(* IEC 61131-3 sources: PortalRobot/Portal_robot/Device/application (part 3) *)

(* ---- PLC_PRG.ReadHmiCommands.st ---- *)
METHOD PRIVATE ReadHmiCommands

// --- BEGIN IMPLEMENTATION ---

// Request counters belong to gateway; pulses and acknowledgements belong to PLC.
udiHmiCommandNowMs := TIME_TO_UDINT(TIME());
GVL_HMI.udiHmiCommandClockMs := udiHmiCommandNowMs;
FOR uiHmiCommandIndex := UINT#1 TO UINT#121 DO
	axHmiCommandConsumed[uiHmiCommandIndex] := FALSE;
	axHmiCommandPulse[uiHmiCommandIndex] := FALSE;
	// Mandatory low scan rearms every existing R_TRIG, including scenario events.
	IF NOT axHmiCommandWasHigh[uiHmiCommandIndex] THEN
		IF axHmiInternalPulse[uiHmiCommandIndex] THEN
			axHmiCommandPulse[uiHmiCommandIndex] := TRUE;
			axHmiInternalPulse[uiHmiCommandIndex] := FALSE;
		ELSE
			audiHmiCommandSnapshot[uiHmiCommandIndex] := GVL_HMI.audiHmiCommandSeq[uiHmiCommandIndex];
			IF (audiHmiCommandSnapshot[uiHmiCommandIndex] <> UDINT#0)
			AND (audiHmiCommandSnapshot[uiHmiCommandIndex] <> GVL_HMI.audiHmiCommandAckSeq[uiHmiCommandIndex]) THEN
				axHmiCommandConsumed[uiHmiCommandIndex] := TRUE;
				IF IsHmiCommandFresh(udiIssuedAtMs := GVL_HMI.audiHmiCommandIssuedAtMs[uiHmiCommandIndex]) THEN
					axHmiCommandPulse[uiHmiCommandIndex] := TRUE;
					GVL_HMI.auiHmiCommandResult[uiHmiCommandIndex] := UINT#1;
				ELSE
					GVL_HMI.auiHmiCommandResult[uiHmiCommandIndex] := UINT#2;
				END_IF;
			END_IF;
		END_IF;
	END_IF;
	axHmiCommandWasHigh[uiHmiCommandIndex] := axHmiCommandPulse[uiHmiCommandIndex];
END_FOR;

// Stable wire IDs; command-contract.mjs and static tests enforce this mapping.
GVL_HMI.xCellEnable := axHmiCommandPulse[1];
GVL_HMI.xCellDisable := axHmiCommandPulse[2];
GVL_HMI.xCellStart := axHmiCommandPulse[3];
GVL_HMI.xCellStop := axHmiCommandPulse[4];
GVL_HMI.xCellReset := axHmiCommandPulse[5];
GVL_HMI.xSafetyRelayReset := axHmiCommandPulse[6];
GVL_HMI.xCellOperatorCancel := axHmiCommandPulse[7];
GVL_HMI.xAlarmResetWarnings := axHmiCommandPulse[8];
GVL_HMI.xModbusSettingsApply := axHmiCommandPulse[9];
GVL_HMI.stMultiType.Command.xAutoDistribute := axHmiCommandPulse[10];
GVL_HMI.xSimAxisGroupError := axHmiCommandPulse[11];
GVL_HMI.xSimRobotWrongAction := axHmiCommandPulse[12];
GVL_HMI.xSimCellBothGrippers := axHmiCommandPulse[13];
GVL_HMI.xSimPointXOutOfLimit := axHmiCommandPulse[14];
GVL_HMI.xSimPointYOutOfLimit := axHmiCommandPulse[15];
GVL_HMI.xSimPointZOutOfLimit := axHmiCommandPulse[16];
GVL_HMI.xSimPointInvalidVelocity := axHmiCommandPulse[17];
GVL_HMI.xSimMagazineWrongOperation := axHmiCommandPulse[18];
GVL_HMI.xSimMagazineNoBlank := axHmiCommandPulse[19];
GVL_HMI.xSimMagazineNoFreeSlot := axHmiCommandPulse[20];
GVL_HMI.xSimMagazineInvalidSlot := axHmiCommandPulse[21];
GVL_HMI.xSimMagazineSlotContent := axHmiCommandPulse[22];
GVL_HMI.xSimMagazineGeometry := axHmiCommandPulse[23];
GVL_HMI.xRobotDrivesEnable := axHmiCommandPulse[24];
GVL_HMI.xRobotDrivesDisable := axHmiCommandPulse[25];
GVL_HMI.xRobotStop := axHmiCommandPulse[26];
GVL_HMI.xRobotReset := axHmiCommandPulse[27];
GVL_HMI.xTestEnvironmentApply := axHmiCommandPulse[28];
GVL_HMI.xTestSpeedProfileApply := axHmiCommandPulse[29];
GVL_HMI.xTestScenarioApply := axHmiCommandPulse[30];
GVL_HMI.xPointCheckStop := axHmiCommandPulse[31];
GVL_HMI.xRobotManualExecute := axHmiCommandPulse[32];
GVL_HMI.stMultiType.Command.xSetTypeCount := axHmiCommandPulse[33];
GVL_HMI.xCellOperatorChoice := axHmiCommandPulse[34];
GVL_HMI.stMultiType.Command.xSetMachineType := axHmiCommandPulse[35];
GVL_HMI.xRobotControlModeApply := axHmiCommandPulse[36];
GVL_HMI.stMultiType.Command.xSetSlotType := axHmiCommandPulse[37];
GVL_HMI.astAxisHmiCommand[1].xHome := axHmiCommandPulse[38];
GVL_HMI.astAxisHmiCommand[1].xMoveAbsolute := axHmiCommandPulse[39];
GVL_HMI.astAxisHmiCommand[1].xMoveRelative := axHmiCommandPulse[40];
GVL_HMI.axSimAxisJogConflict[1] := axHmiCommandPulse[41];
GVL_HMI.axMachineSimReset[1] := axHmiCommandPulse[42];
GVL_HMI.axMachineEnable[1] := axHmiCommandPulse[43];
GVL_HMI.axMachineDisable[1] := axHmiCommandPulse[44];
GVL_HMI.axMachineReset[1] := axHmiCommandPulse[45];
GVL_HMI.axMachineSetBlank[1] := axHmiCommandPulse[46];
GVL_HMI.axMachineSetDetail[1] := axHmiCommandPulse[47];
GVL_HMI.axMachineAcceptDoor[1] := axHmiCommandPulse[48];
GVL_HMI.axMachineRejectDoor[1] := axHmiCommandPulse[49];
GVL_HMI.axMachineAcceptRun[1] := axHmiCommandPulse[50];
GVL_HMI.axMachineRejectRun[1] := axHmiCommandPulse[51];
GVL_HMI.axMachineManualSafetyDoorOpen[1] := axHmiCommandPulse[52];
GVL_HMI.axMachineManualSafetyDoorClose[1] := axHmiCommandPulse[53];
GVL_HMI.axMachineManualHatchOpen[1] := axHmiCommandPulse[54];
GVL_HMI.axMachineManualHatchClose[1] := axHmiCommandPulse[55];
GVL_HMI.axMachineManualHatchUnlock[1] := axHmiCommandPulse[56];
GVL_HMI.axMachineManualHatchLock[1] := axHmiCommandPulse[57];
GVL_HMI.axMachineManualChuckOpen[1] := axHmiCommandPulse[58];
GVL_HMI.axMachineManualChuckClose[1] := axHmiCommandPulse[59];
GVL_HMI.astAxisHmiCommand[2].xHome := axHmiCommandPulse[60];
GVL_HMI.astAxisHmiCommand[2].xMoveAbsolute := axHmiCommandPulse[61];
GVL_HMI.astAxisHmiCommand[2].xMoveRelative := axHmiCommandPulse[62];
GVL_HMI.axSimAxisJogConflict[2] := axHmiCommandPulse[63];
GVL_HMI.axMachineSimReset[2] := axHmiCommandPulse[64];
GVL_HMI.axMachineEnable[2] := axHmiCommandPulse[65];
GVL_HMI.axMachineDisable[2] := axHmiCommandPulse[66];
GVL_HMI.axMachineReset[2] := axHmiCommandPulse[67];
GVL_HMI.axMachineSetBlank[2] := axHmiCommandPulse[68];
GVL_HMI.axMachineSetDetail[2] := axHmiCommandPulse[69];
GVL_HMI.axMachineAcceptDoor[2] := axHmiCommandPulse[70];
GVL_HMI.axMachineRejectDoor[2] := axHmiCommandPulse[71];
GVL_HMI.axMachineAcceptRun[2] := axHmiCommandPulse[72];
GVL_HMI.axMachineRejectRun[2] := axHmiCommandPulse[73];
GVL_HMI.axMachineManualSafetyDoorOpen[2] := axHmiCommandPulse[74];
GVL_HMI.axMachineManualSafetyDoorClose[2] := axHmiCommandPulse[75];
GVL_HMI.axMachineManualHatchOpen[2] := axHmiCommandPulse[76];
GVL_HMI.axMachineManualHatchClose[2] := axHmiCommandPulse[77];
GVL_HMI.axMachineManualHatchUnlock[2] := axHmiCommandPulse[78];
GVL_HMI.axMachineManualHatchLock[2] := axHmiCommandPulse[79];
GVL_HMI.axMachineManualChuckOpen[2] := axHmiCommandPulse[80];
GVL_HMI.axMachineManualChuckClose[2] := axHmiCommandPulse[81];
GVL_HMI.astAxisHmiCommand[3].xHome := axHmiCommandPulse[82];
GVL_HMI.astAxisHmiCommand[3].xMoveAbsolute := axHmiCommandPulse[83];
GVL_HMI.astAxisHmiCommand[3].xMoveRelative := axHmiCommandPulse[84];
GVL_HMI.axSimAxisJogConflict[3] := axHmiCommandPulse[85];
GVL_HMI.axMachineSimReset[3] := axHmiCommandPulse[86];
GVL_HMI.axMachineEnable[3] := axHmiCommandPulse[87];
GVL_HMI.axMachineDisable[3] := axHmiCommandPulse[88];
GVL_HMI.axMachineReset[3] := axHmiCommandPulse[89];
GVL_HMI.axMachineSetBlank[3] := axHmiCommandPulse[90];
GVL_HMI.axMachineSetDetail[3] := axHmiCommandPulse[91];
GVL_HMI.axMachineAcceptDoor[3] := axHmiCommandPulse[92];
GVL_HMI.axMachineRejectDoor[3] := axHmiCommandPulse[93];
GVL_HMI.axMachineAcceptRun[3] := axHmiCommandPulse[94];
GVL_HMI.axMachineRejectRun[3] := axHmiCommandPulse[95];
GVL_HMI.axMachineManualSafetyDoorOpen[3] := axHmiCommandPulse[96];
GVL_HMI.axMachineManualSafetyDoorClose[3] := axHmiCommandPulse[97];
GVL_HMI.axMachineManualHatchOpen[3] := axHmiCommandPulse[98];
GVL_HMI.axMachineManualHatchClose[3] := axHmiCommandPulse[99];
GVL_HMI.axMachineManualHatchUnlock[3] := axHmiCommandPulse[100];
GVL_HMI.axMachineManualHatchLock[3] := axHmiCommandPulse[101];
GVL_HMI.axMachineManualChuckOpen[3] := axHmiCommandPulse[102];
GVL_HMI.axMachineManualChuckClose[3] := axHmiCommandPulse[103];
GVL_HMI.astMagazineCommand[1].xEnable := axHmiCommandPulse[104];
GVL_HMI.astMagazineCommand[1].xDisable := axHmiCommandPulse[105];
GVL_HMI.astMagazineCommand[1].xStop := axHmiCommandPulse[106];
GVL_HMI.astMagazineCommand[1].xReset := axHmiCommandPulse[107];
GVL_HMI.astMagazineCommand[1].xFill := axHmiCommandPulse[108];
GVL_HMI.astMagazineCommand[1].xClear := axHmiCommandPulse[109];
GVL_HMI.astMagazineCommand[1].xApplySlot := axHmiCommandPulse[110];
GVL_HMI.astMagazineCommand[1].xApplyPitchX := axHmiCommandPulse[111];
GVL_HMI.astMagazineCommand[1].xApplyPitchY := axHmiCommandPulse[112];
GVL_HMI.astMagazineCommand[2].xEnable := axHmiCommandPulse[113];
GVL_HMI.astMagazineCommand[2].xDisable := axHmiCommandPulse[114];
GVL_HMI.astMagazineCommand[2].xStop := axHmiCommandPulse[115];
GVL_HMI.astMagazineCommand[2].xReset := axHmiCommandPulse[116];
GVL_HMI.astMagazineCommand[2].xFill := axHmiCommandPulse[117];
GVL_HMI.astMagazineCommand[2].xClear := axHmiCommandPulse[118];
GVL_HMI.astMagazineCommand[2].xApplySlot := axHmiCommandPulse[119];
GVL_HMI.astMagazineCommand[2].xApplyPitchX := axHmiCommandPulse[120];
GVL_HMI.astMagazineCommand[2].xApplyPitchY := axHmiCommandPulse[121];

(* ---- PLC_PRG.ReadHmiInputs.st ---- *)
METHOD PRIVATE ReadHmiInputs

// --- BEGIN IMPLEMENTATION ---

// HMI обязана поддерживать heartbeat. При потере связи PLC снимает только
// расширенные ручные команды; технологические проверки ниже остаются в PLC.
tonHmiWatchdog(
	IN := GVL_HMI.udiHmiHeartbeat = udiLastHmiHeartbeat,
	PT := T#2S
);
IF GVL_HMI.udiHmiHeartbeat <> udiLastHmiHeartbeat THEN
	udiLastHmiHeartbeat := GVL_HMI.udiHmiHeartbeat;
END_IF;
xHmiConnectionAlive := NOT tonHmiWatchdog.Q;

// Мобильная аренда отделена от общего HMI heartbeat. Gateway может быть жив,
// но движение обязано остановиться, если телефон перестал подтверждать аренду.
rtMobileMotionStart(CLK := GVL_HMI.xMobileMotionActive);
tonMobileMotionWatchdog(
	IN := GVL_HMI.xMobileMotionActive
		AND (GVL_HMI.udiMobileMotionHeartbeat = udiLastMobileMotionHeartbeat),
	PT := T#2S
);
IF GVL_HMI.udiMobileMotionHeartbeat <> udiLastMobileMotionHeartbeat THEN
	udiLastMobileMotionHeartbeat := GVL_HMI.udiMobileMotionHeartbeat;
END_IF;
IF rtMobileMotionStart.Q THEN
	xMobileMotionLeaseActive := TRUE;
	rMobileMotionSpeedLimitPercent := LIMIT(
		REAL#0.1,
		GVL_CELL_SETTINGS.rPointCheckSpeedPercent,
		REAL#100.0
	);
END_IF;
IF xMobileMotionLeaseActive THEN
	// Во время аренды лимит разрешено только уменьшать. Повышение настройки
	// применяется уже к следующему мобильному движению.
	rMobileMotionSpeedLimitPercent := MIN(
		rMobileMotionSpeedLimitPercent,
		LIMIT(REAL#0.1, GVL_CELL_SETTINGS.rPointCheckSpeedPercent, REAL#100.0)
	);
END_IF;
xMobileMotionConnectionAlive := GVL_HMI.xMobileMotionActive
	AND NOT tonMobileMotionWatchdog.Q;
xMobileMotionStopRequest := xMobileMotionLeaseActive
	AND (NOT GVL_HMI.xMobileMotionActive
		OR NOT xMobileMotionConnectionAlive
		OR NOT xHmiConnectionAlive);
IF xMobileMotionStopRequest THEN
	// Сбрасываем вход аренды в PLC: восстановление сети не может само возобновить ход.
	GVL_HMI.xMobileMotionActive := FALSE;
	FOR uiMachine := 1 TO 3 DO
		GVL_HMI.astAxisHmiCommand[uiMachine].xJogPositive := FALSE;
		GVL_HMI.astAxisHmiCommand[uiMachine].xJogNegative := FALSE;
	END_FOR;
END_IF;
GVL_HMI.xMobileMotionLeaseAlive := xMobileMotionLeaseActive
	AND xMobileMotionConnectionAlive
	AND NOT xMobileMotionStopRequest;
GVL_HMI.rMobileMotionAppliedSpeedPercent := rMobileMotionSpeedLimitPercent;

xPointCheckRequest := FALSE;
tonPointCheckWatchdog(IN := GVL_HMI.udiPointCheckHeartbeat = udiLastPointCheckHeartbeat, PT := T#2S);
IF GVL_HMI.udiPointCheckHeartbeat <> udiLastPointCheckHeartbeat THEN
	udiLastPointCheckHeartbeat := GVL_HMI.udiPointCheckHeartbeat;
END_IF;
xPointCheckConnectionAlive := (udiLastPointCheckHeartbeat <> UDINT#0) AND NOT tonPointCheckWatchdog.Q;
xPointCheckStopRequest := xPointCheckActive AND (GVL_HMI.xPointCheckStop
	OR NOT xPointCheckConnectionAlive OR NOT xHmiConnectionAlive);
// Stop is a PLC-owned one-scan event; its request counter is never cleared here.

IF GVL_HMI.rRobotManualSpeedPercent < REAL#0.1 THEN
	GVL_HMI.rRobotManualSpeedPercent := REAL#0.1;
ELSIF GVL_HMI.rRobotManualSpeedPercent > REAL#100.0 THEN
	GVL_HMI.rRobotManualSpeedPercent := REAL#100.0;
END_IF;
IF (GVL_HMI.lrRobotManualStep <> 0.1)
AND (GVL_HMI.lrRobotManualStep <> 1.0)
AND (GVL_HMI.lrRobotManualStep <> 10.0)
AND (GVL_HMI.lrRobotManualStep <> 100.0) THEN
	GVL_HMI.lrRobotManualStep := 1.0;
END_IF;

IF NOT xHmiConnectionAlive THEN
	FOR uiMachine := 1 TO 3 DO
		GVL_HMI.astAxisHmiCommand[uiMachine].xJogPositive := FALSE;
		GVL_HMI.astAxisHmiCommand[uiMachine].xJogNegative := FALSE;
		GVL_HMI.astAxisHmiCommand[uiMachine].xHome := FALSE;
		GVL_HMI.astAxisHmiCommand[uiMachine].xMoveAbsolute := FALSE;
		GVL_HMI.astAxisHmiCommand[uiMachine].xMoveRelative := FALSE;
	END_FOR;
	FOR uiMagazine := UINT#1 TO UINT#2 DO
		GVL_HMI.astMagazineCommand[uiMagazine].xStop := FALSE;
	END_FOR;
	GVL_HMI.xRobotManualExecute := FALSE;
END_IF;

// Глобальные команды ячейки поступают через единый интерфейс HMI.
GVL_CELL_CONTROL.xEnable := GVL_HMI.xCellEnable;
GVL_CELL_CONTROL.xDisable := GVL_HMI.xCellDisable;
GVL_CELL_CONTROL.xStart := GVL_HMI.xCellStart;
GVL_CELL_CONTROL.xStop := GVL_HMI.xCellStop;
// Необработанный общий импульс передаётся всем владельцам аварий.
// Каждый функциональный блок самостоятельно проверяет возможность сброса.
GVL_CELL_CONTROL.xReset := GVL_HMI.xCellReset;
// Режим хранит PLC. Новая транзакция применяется в RunSafety после чтения
// актуальных входов безопасности; PublishHmi не пишет в буфер запроса.
GVL_ALARM.Command.xResetWarnings := GVL_HMI.xAlarmResetWarnings;

// Режим инъекции ошибок включается отдельным переключателем страницы CELL_SETTINGS.
GVL_CELL_SETTINGS.xErrorSimulationEnabled := GVL_HMI.xErrorSimulationEnable;

// Ползунок меняет только запрошенное значение. Отдельный FB применяет его к
// таймерам и Dynamic Limits безопасной транзакцией перед следующим тестом.
GVL_CELL_SETTINGS.xSimulationAccelerationChangeAllowed :=
	xHmiConnectionAlive
	AND NOT GVL_CELL_CONTROL.xGlobalError;

IF GVL_CELL_SETTINGS.xSimulationAccelerationChangeAllowed THEN
	GVL_CELL_SETTINGS.xSimulationAccelerationEnable := GVL_HMI.xSimulationAccelerationEnable;
	GVL_CELL_SETTINGS.uiSimulationTimeFactor := GVL_HMI.uiSimulationTimeFactor;
	IF GVL_CELL_SETTINGS.uiSimulationTimeFactor < UINT#1 THEN
		GVL_CELL_SETTINGS.uiSimulationTimeFactor := UINT#1;
	ELSIF GVL_CELL_SETTINGS.uiSimulationTimeFactor > UINT#100 THEN
		GVL_CELL_SETTINGS.uiSimulationTimeFactor := UINT#100;
	END_IF;
ELSE
	// При потере разрешения сохраняем последнее принятое требование.
	GVL_HMI.xSimulationAccelerationEnable := GVL_CELL_SETTINGS.xSimulationAccelerationActive;
	GVL_HMI.uiSimulationTimeFactor := GVL_CELL_SETTINGS.uiSimulationTimeFactor;
END_IF;

// Общие технологические TIMEOUT и допуски HOME принимаются только при полностью
// остановленной ячейке. Координатами HOME_SAFETY владеет редактор точек ниже.
GVL_CELL_SETTINGS.xCellSettingsChangeAllowed :=
	xHmiConnectionAlive
	AND NOT GVL_CELL_MANAGER.Status.xRunning
	AND NOT GVL_HMI.xModbusMode
	AND NOT GVL_CELL_CONTROL.xGlobalError
	AND NOT GVL_AXIS.arrAxis[1].Status.xMotionBusy
	AND NOT GVL_AXIS.arrAxis[2].Status.xMotionBusy
	AND NOT GVL_AXIS.arrAxis[3].Status.xMotionBusy
	AND NOT GVL_AXIS_GROUP.AxisGroup.Command.xMoveDirect
	AND NOT GVL_AXIS_GROUP.AxisGroup.Command.xMoveLinear
	AND NOT GVL_ROBOT.Status.xBusy;

// Independent requested value; publication cannot overwrite an incoming write.
xCellSettingRejected := FALSE;
udiCellSettingSnapshot := GVL_HMI.udiCellSettingCommandSeq;
IF (udiCellSettingSnapshot <> UDINT#0)
AND (udiCellSettingSnapshot <> GVL_HMI.udiCellSettingAckSeq) THEN
	GVL_HMI.uiCellSettingResult := UINT#3;
	IF NOT IsHmiCommandFresh(udiIssuedAtMs := GVL_HMI.udiCellSettingIssuedAtMs) THEN
		GVL_HMI.uiCellSettingResult := UINT#4; // Expired: never apply later
	ELSIF NOT GVL_CELL_SETTINGS.xCellSettingsChangeAllowed
	OR ((GVL_HMI.uiCellSettingIndex = UINT#4) AND xPointCheckActive) THEN
		GVL_HMI.uiCellSettingResult := UINT#2;
	ELSE
		CASE GVL_HMI.uiCellSettingIndex OF
			UINT#1:
				IF (GVL_HMI.lrCellSettingRequest >= 0.1) AND (GVL_HMI.lrCellSettingRequest <= 1000.0) THEN
					GVL_CELL_SETTINGS.lrSafetyHomeToleranceX := GVL_HMI.lrCellSettingRequest;
					GVL_HMI.uiCellSettingResult := UINT#1;
				END_IF;
			UINT#2:
				IF (GVL_HMI.lrCellSettingRequest >= 0.1) AND (GVL_HMI.lrCellSettingRequest <= 1000.0) THEN
					GVL_CELL_SETTINGS.lrSafetyHomeToleranceY := GVL_HMI.lrCellSettingRequest;
					GVL_HMI.uiCellSettingResult := UINT#1;
				END_IF;
			UINT#3:
				IF (GVL_HMI.lrCellSettingRequest >= 0.1) AND (GVL_HMI.lrCellSettingRequest <= 1000.0) THEN
					GVL_CELL_SETTINGS.lrSafetyHomeToleranceZ := GVL_HMI.lrCellSettingRequest;
					GVL_HMI.uiCellSettingResult := UINT#1;
				END_IF;
			UINT#4:
				IF (GVL_HMI.lrCellSettingRequest >= 0.1) AND (GVL_HMI.lrCellSettingRequest <= 100.0) THEN
					GVL_CELL_SETTINGS.rPointCheckSpeedPercent := LREAL_TO_REAL(GVL_HMI.lrCellSettingRequest);
					GVL_HMI.uiCellSettingResult := UINT#1;
				END_IF;
			UINT#5:
				IF (GVL_HMI.lrCellSettingRequest >= 1000.0) AND (GVL_HMI.lrCellSettingRequest <= 600000.0) THEN
					GVL_CELL_SETTINGS.stMachineTimeouts.tRobotMove := UDINT_TO_TIME(LREAL_TO_UDINT(GVL_HMI.lrCellSettingRequest));
					GVL_HMI.uiCellSettingResult := UINT#1;
				END_IF;
			UINT#6:
				IF (GVL_HMI.lrCellSettingRequest >= 1000.0) AND (GVL_HMI.lrCellSettingRequest <= 600000.0) THEN
					GVL_CELL_SETTINGS.stMachineTimeouts.tRobotAction := UDINT_TO_TIME(LREAL_TO_UDINT(GVL_HMI.lrCellSettingRequest));
					GVL_HMI.uiCellSettingResult := UINT#1;
				END_IF;
			UINT#7:
				IF (GVL_HMI.lrCellSettingRequest >= 1000.0) AND (GVL_HMI.lrCellSettingRequest <= 600000.0) THEN
					GVL_CELL_SETTINGS.stMachineTimeouts.tRobotRelease := UDINT_TO_TIME(LREAL_TO_UDINT(GVL_HMI.lrCellSettingRequest));
					GVL_HMI.uiCellSettingResult := UINT#1;
				END_IF;
			UINT#8:
				IF (GVL_HMI.lrCellSettingRequest >= 1000.0) AND (GVL_HMI.lrCellSettingRequest <= 600000.0) THEN
					GVL_CELL_SETTINGS.stMachineTimeouts.tDoorOpen := UDINT_TO_TIME(LREAL_TO_UDINT(GVL_HMI.lrCellSettingRequest));
					GVL_HMI.uiCellSettingResult := UINT#1;
				END_IF;
			UINT#9:
				IF (GVL_HMI.lrCellSettingRequest >= 1000.0) AND (GVL_HMI.lrCellSettingRequest <= 600000.0) THEN
					GVL_CELL_SETTINGS.stMachineTimeouts.tDoorClose := UDINT_TO_TIME(LREAL_TO_UDINT(GVL_HMI.lrCellSettingRequest));
					GVL_HMI.uiCellSettingResult := UINT#1;
				END_IF;
			UINT#10:
				IF (GVL_HMI.lrCellSettingRequest >= 1000.0) AND (GVL_HMI.lrCellSettingRequest <= 600000.0) THEN
					GVL_CELL_SETTINGS.stMachineTimeouts.tHatchUnlock := UDINT_TO_TIME(LREAL_TO_UDINT(GVL_HMI.lrCellSettingRequest));
					GVL_HMI.uiCellSettingResult := UINT#1;
				END_IF;
			UINT#11:
				IF (GVL_HMI.lrCellSettingRequest >= 1000.0) AND (GVL_HMI.lrCellSettingRequest <= 600000.0) THEN
					GVL_CELL_SETTINGS.stMachineTimeouts.tChuckOpen := UDINT_TO_TIME(LREAL_TO_UDINT(GVL_HMI.lrCellSettingRequest));
					GVL_HMI.uiCellSettingResult := UINT#1;
				END_IF;
			UINT#12:
				IF (GVL_HMI.lrCellSettingRequest >= 1000.0) AND (GVL_HMI.lrCellSettingRequest <= 600000.0) THEN
					GVL_CELL_SETTINGS.stMachineTimeouts.tChuckClose := UDINT_TO_TIME(LREAL_TO_UDINT(GVL_HMI.lrCellSettingRequest));
					GVL_HMI.uiCellSettingResult := UINT#1;
				END_IF;
			UINT#13:
				IF (GVL_HMI.lrCellSettingRequest >= 1000.0) AND (GVL_HMI.lrCellSettingRequest <= 600000.0) THEN
					GVL_CELL_SETTINGS.stMachineTimeouts.tCycleStart := UDINT_TO_TIME(LREAL_TO_UDINT(GVL_HMI.lrCellSettingRequest));
					GVL_HMI.uiCellSettingResult := UINT#1;
				END_IF;
		END_CASE;
	END_IF;
	xCellSettingRejected := GVL_HMI.uiCellSettingResult <> UINT#1;
END_IF;

// =============================================================================
// Транзакционный редактор 12 фиксированных инженерных точек
// =============================================================================
xPointEditorAllHomed := GVL_AXIS.arrAxis[1].Status.xHomed
	AND GVL_AXIS.arrAxis[2].Status.xHomed
	AND GVL_AXIS.arrAxis[3].Status.xHomed;
xPointEditorBaseAllowed := xHmiConnectionAlive
	AND NOT xPointCheckActive
	AND GVL_CELL_CONTROL.xManual
	AND NOT GVL_HMI.xModbusMode
	AND NOT GVL_CELL_MANAGER.Status.xRunning
	AND NOT GVL_CELL_CONTROL.xGlobalError
	AND NOT GVL_ROBOT.Status.xBusy
	AND NOT xMotionBusy
	AND NOT xDriveError
	AND NOT GVL_MOTION_MANAGER.stMotionManager.Status.xError
	AND xPointEditorAllHomed
	AND GVL_AXIS_GROUP.AxisGroup.Status.xPositionValid;
GVL_HMI.xPointEditorCaptureAllowed := xPointEditorBaseAllowed;
GVL_HMI.xPointEditorSaveAllowed := xPointEditorBaseAllowed
	AND GVL_POINT_MANAGER.PointManager.Diag.xXLimitValid
	AND GVL_POINT_MANAGER.PointManager.Diag.xYLimitValid
	AND GVL_POINT_MANAGER.PointManager.Diag.xZLimitValid;

IF (GVL_HMI.udiPointEditorCommandSeq <> UDINT#0)
AND (GVL_HMI.udiPointEditorCommandSeq <> udiLastPointEditorCommandSeq) THEN
	udiLastPointEditorCommandSeq := GVL_HMI.udiPointEditorCommandSeq;
	GVL_HMI.uiPointEditorResult := UINT#2;
	GVL_HMI.uiPointEditorRejectReason := UINT#0;
	xPointEditorRequestValid := FALSE;
	xPointEditorMagazinePoint := FALSE;
	ePointEditorName := E_POINT_NAME.NONE;
	uiPointStorageIndex := UINT#0;

	CASE GVL_HMI.uiPointEditorIndex OF
		UINT#1: ePointEditorName := E_POINT_NAME.MACHINE_1_ABOVE; uiPointStorageIndex := UINT#1;
		UINT#2: ePointEditorName := E_POINT_NAME.MACHINE_1_CHUCK_APROACH; uiPointStorageIndex := UINT#3;
		UINT#3: ePointEditorName := E_POINT_NAME.MACHINE_1_CHUCK_POSITION; uiPointStorageIndex := UINT#4;
		UINT#4: ePointEditorName := E_POINT_NAME.MACHINE_2_ABOVE; uiPointStorageIndex := UINT#5;
		UINT#5: ePointEditorName := E_POINT_NAME.MACHINE_2_CHUCK_APROACH; uiPointStorageIndex := UINT#7;
		UINT#6: ePointEditorName := E_POINT_NAME.MACHINE_2_CHUCK_POSITION; uiPointStorageIndex := UINT#8;
		UINT#7: ePointEditorName := E_POINT_NAME.MACHINE_3_ABOVE; uiPointStorageIndex := UINT#9;
		UINT#8: ePointEditorName := E_POINT_NAME.MACHINE_3_CHUCK_APROACH; uiPointStorageIndex := UINT#11;
		UINT#9: ePointEditorName := E_POINT_NAME.MACHINE_3_CHUCK_POSITION; uiPointStorageIndex := UINT#12;
		UINT#10: ePointEditorName := E_POINT_NAME.HOME_SAFETY; uiPointStorageIndex := UINT#13;
		UINT#11: ePointEditorName := E_POINT_NAME.MAGAZINE_1_DETAIL; uiPointStorageIndex := UINT#14;
		UINT#12: ePointEditorName := E_POINT_NAME.MAGAZINE_2_DETAIL; uiPointStorageIndex := UINT#15;
	END_CASE;
	xPointEditorRequestValid := (ePointEditorName <> E_POINT_NAME.NONE)
		AND (uiPointStorageIndex <> UINT#0);
	xPointEditorMagazinePoint := (ePointEditorName = E_POINT_NAME.MAGAZINE_1_DETAIL)
		OR (ePointEditorName = E_POINT_NAME.MAGAZINE_2_DETAIL);

	IF (GVL_HMI.uiPointEditorCommand <> UINT#1)
	AND (GVL_HMI.uiPointEditorCommand <> UINT#2)
	AND (GVL_HMI.uiPointEditorCommand <> UINT#3) THEN
		GVL_HMI.uiPointEditorRejectReason := UINT#1; // Неизвестная команда
	ELSIF NOT xPointEditorRequestValid THEN
		GVL_HMI.uiPointEditorRejectReason := UINT#2; // Неверный индекс точки
	ELSIF NOT xHmiConnectionAlive THEN
		GVL_HMI.uiPointEditorRejectReason := UINT#3; // HMI offline
	ELSIF NOT GVL_CELL_CONTROL.xManual THEN
		GVL_HMI.uiPointEditorRejectReason := UINT#4; // Требуется ручной режим
	ELSIF GVL_HMI.xModbusMode THEN
		GVL_HMI.uiPointEditorRejectReason := UINT#5; // Требуется SoftMotion
	ELSIF GVL_CELL_MANAGER.Status.xRunning THEN
		GVL_HMI.uiPointEditorRejectReason := UINT#6; // Автоматический цикл выполняется
	ELSIF GVL_CELL_CONTROL.xGlobalError THEN
		GVL_HMI.uiPointEditorRejectReason := UINT#7; // Глобальная ошибка
	ELSIF GVL_ROBOT.Status.xBusy OR xPointCheckActive THEN
		GVL_HMI.uiPointEditorRejectReason := UINT#8; // Робот занят
	ELSIF xMotionBusy THEN
		GVL_HMI.uiPointEditorRejectReason := UINT#9; // Motion занят
	ELSIF xDriveError OR GVL_MOTION_MANAGER.stMotionManager.Status.xError THEN
		GVL_HMI.uiPointEditorRejectReason := UINT#10; // Ошибка оси или группы
	ELSIF NOT xPointEditorAllHomed THEN
		GVL_HMI.uiPointEditorRejectReason := UINT#11; // Не выполнен Home
	ELSIF NOT GVL_AXIS_GROUP.AxisGroup.Status.xPositionValid THEN
		GVL_HMI.uiPointEditorRejectReason := UINT#12; // Недостоверные координаты
	ELSIF (GVL_HMI.uiPointEditorCommand = UINT#2)
	AND (NOT GVL_POINT_MANAGER.PointManager.Diag.xXLimitValid
		OR NOT GVL_POINT_MANAGER.PointManager.Diag.xYLimitValid
		OR NOT GVL_POINT_MANAGER.PointManager.Diag.xZLimitValid) THEN
		GVL_HMI.uiPointEditorRejectReason := UINT#13; // Software limits недоступны
	ELSE
		IF GVL_HMI.uiPointEditorCommand = UINT#1 THEN
			// CAPTURE возвращает согласованный снимок одного PLC-цикла и не пишет Persistent.
			GVL_HMI.stPointEditorResultPoint.Name := '';
			GVL_HMI.stPointEditorResultPoint.X := GVL_AXIS_GROUP.AxisGroup.Status.ActualX;
			GVL_HMI.stPointEditorResultPoint.Y := GVL_AXIS_GROUP.AxisGroup.Status.ActualY;
			GVL_HMI.stPointEditorResultPoint.Z := GVL_AXIS_GROUP.AxisGroup.Status.ActualZ;
			GVL_HMI.stPointEditorResultPoint.MagazineSafeZ :=
				GVL_HMI.lrPointEditorDraftMagazineSafeZ;
			GVL_HMI.stPointEditorResultPoint.MagazineChangeZ :=
				GVL_HMI.lrPointEditorDraftMagazineChangeZ;
			GVL_HMI.stPointEditorResultPoint.SpeedFactor :=
				GVL_HMI.lrPointEditorDraftSpeedFactor;
			GVL_HMI.stPointEditorResultPoint.xConfigured := FALSE;
			GVL_HMI.uiPointEditorResult := UINT#1;
		ELSIF GVL_HMI.uiPointEditorCommand = UINT#3 THEN
			// CHECK никогда не сохраняет черновик. Сравнение защищает подтверждение
			// на телефоне от изменения точки другим редактором до запуска.
			IF NOT GVL_POINT.Points[ePointEditorName].xConfigured THEN
				GVL_HMI.uiPointEditorRejectReason := UINT#16;
			ELSIF (GVL_POINT.Points[ePointEditorName].X <> GVL_HMI.alrPointEditorDraftXYZ[1])
			OR (GVL_POINT.Points[ePointEditorName].Y <> GVL_HMI.alrPointEditorDraftXYZ[2])
			OR (GVL_POINT.Points[ePointEditorName].Z <> GVL_HMI.alrPointEditorDraftXYZ[3])
			OR (GVL_POINT.Points[ePointEditorName].SpeedFactor <> GVL_HMI.lrPointEditorDraftSpeedFactor)
			OR (xPointEditorMagazinePoint
				AND ((GVL_POINT.Points[ePointEditorName].MagazineSafeZ <>
					GVL_HMI.lrPointEditorDraftMagazineSafeZ)
				OR (GVL_POINT.Points[ePointEditorName].MagazineChangeZ <>
					GVL_HMI.lrPointEditorDraftMagazineChangeZ))) THEN
				GVL_HMI.uiPointEditorRejectReason := UINT#21;
			ELSE
				xPointCheckRequest := TRUE; // Финальное разрешение после RunMotion/RunCellControl
			END_IF;
		ELSE
			xPointEditorDraftValid :=
				(GVL_HMI.alrPointEditorDraftXYZ[1] >= alrRobotSoftwareMinPosition[1])
				AND (GVL_HMI.alrPointEditorDraftXYZ[1] <= alrRobotSoftwareMaxPosition[1])
				AND (GVL_HMI.alrPointEditorDraftXYZ[2] >= alrRobotSoftwareMinPosition[2])
				AND (GVL_HMI.alrPointEditorDraftXYZ[2] <= alrRobotSoftwareMaxPosition[2])
				AND (GVL_HMI.alrPointEditorDraftXYZ[3] >= alrRobotSoftwareMinPosition[3])
				AND (GVL_HMI.alrPointEditorDraftXYZ[3] <= alrRobotSoftwareMaxPosition[3]);
			IF NOT xPointEditorDraftValid THEN
				GVL_HMI.uiPointEditorRejectReason := UINT#14; // XYZ вне software limits
			ELSIF NOT ((GVL_HMI.lrPointEditorDraftSpeedFactor > 0.1)
			AND (GVL_HMI.lrPointEditorDraftSpeedFactor <= 1.0)) THEN
				GVL_HMI.uiPointEditorRejectReason := UINT#15; // Недопустимая скорость
			ELSIF xPointEditorMagazinePoint
			AND ((GVL_HMI.lrPointEditorDraftMagazineSafeZ < -LREAL#10000.0)
				OR (GVL_HMI.lrPointEditorDraftMagazineSafeZ > LREAL#10000.0)
				OR (GVL_HMI.lrPointEditorDraftMagazineChangeZ < -LREAL#10000.0)
				OR (GVL_HMI.lrPointEditorDraftMagazineChangeZ > LREAL#10000.0)) THEN
				GVL_HMI.uiPointEditorRejectReason := UINT#22; // Смещения магазина вне диапазона
			ELSE
				GVL_POINT.astRetainPoints[uiPointStorageIndex].Name := '';
				GVL_POINT.astRetainPoints[uiPointStorageIndex].X :=
					GVL_HMI.alrPointEditorDraftXYZ[1];
				GVL_POINT.astRetainPoints[uiPointStorageIndex].Y :=
					GVL_HMI.alrPointEditorDraftXYZ[2];
				GVL_POINT.astRetainPoints[uiPointStorageIndex].Z :=
					GVL_HMI.alrPointEditorDraftXYZ[3];
				IF xPointEditorMagazinePoint THEN
					GVL_POINT.astRetainPoints[uiPointStorageIndex].MagazineSafeZ :=
						GVL_HMI.lrPointEditorDraftMagazineSafeZ;
					GVL_POINT.astRetainPoints[uiPointStorageIndex].MagazineChangeZ :=
						GVL_HMI.lrPointEditorDraftMagazineChangeZ;
				ELSE
					GVL_POINT.astRetainPoints[uiPointStorageIndex].MagazineSafeZ := LREAL#0.0;
					GVL_POINT.astRetainPoints[uiPointStorageIndex].MagazineChangeZ := LREAL#0.0;
				END_IF;
				GVL_POINT.astRetainPoints[uiPointStorageIndex].SpeedFactor :=
					GVL_HMI.lrPointEditorDraftSpeedFactor;
				GVL_POINT.astRetainPoints[uiPointStorageIndex].xConfigured :=
					NOT xPointEditorMagazinePoint
					OR ((GVL_HMI.lrPointEditorDraftMagazineSafeZ <> LREAL#0.0)
						AND (GVL_HMI.lrPointEditorDraftMagazineChangeZ <> LREAL#0.0));
				GVL_POINT.Points[ePointEditorName] :=
					GVL_POINT.astRetainPoints[uiPointStorageIndex];
				GVL_HMI.stPointEditorResultPoint := GVL_POINT.Points[ePointEditorName];
				GVL_HMI.uiPointEditorResult := UINT#1;
			END_IF;
		END_IF;
	END_IF;

	IF (GVL_HMI.uiPointEditorResult <> UINT#1) AND NOT xPointCheckRequest THEN
		IF GVL_HMI.uiPointEditorCommand = UINT#3 THEN
			uiRobotInterfaceWarningCode := WRN_POINT_CHECK_REJECTED;
		ELSE
			uiRobotInterfaceWarningCode := WRN_POINT_EDIT_REJECTED;
		END_IF;
	END_IF;
	// Ack подтверждает обработку конкретной транзакции даже при отказе.
	IF NOT xPointCheckRequest THEN
		GVL_HMI.udiPointEditorAckSeq := GVL_HMI.udiPointEditorCommandSeq;
	END_IF;
END_IF;

// Плоский OPC UA-интерфейс HMI преобразуется в типизированные запросы FB.
FOR uiMachine := 1 TO 3 DO
	astMachineFaultRequest[uiMachine].xEnabled := GVL_CELL_SETTINGS.xErrorSimulationEnabled;
	astMachineFaultRequest[uiMachine].xReset := GVL_HMI.axMachineSimReset[uiMachine];
	astMachineFaultRequest[uiMachine].xMachineAlarm := GVL_HMI.axMachineSimAlarm[uiMachine];
	astMachineFaultRequest[uiMachine].xDoorFault := GVL_HMI.axMachineSimDoorFault[uiMachine];
	astMachineFaultRequest[uiMachine].xChuckFault := GVL_HMI.axMachineSimChuckFault[uiMachine];
	astMachineFaultRequest[uiMachine].xTimeoutRobotMove := GVL_HMI.axMachineTimeoutRobotMove[uiMachine];
	astMachineFaultRequest[uiMachine].xTimeoutRobotAction := GVL_HMI.axMachineTimeoutRobotAction[uiMachine];
	astMachineFaultRequest[uiMachine].xTimeoutRobotRelease := GVL_HMI.axMachineTimeoutRobotRelease[uiMachine];
	astMachineFaultRequest[uiMachine].xTimeoutDoorOpen := GVL_HMI.axMachineTimeoutDoorOpen[uiMachine];
	astMachineFaultRequest[uiMachine].xTimeoutDoorClose := GVL_HMI.axMachineTimeoutDoorClose[uiMachine];
	astMachineFaultRequest[uiMachine].xTimeoutHatchUnlock := GVL_HMI.axMachineTimeoutHatchUnlock[uiMachine];
	astMachineFaultRequest[uiMachine].xTimeoutChuckOpen := GVL_HMI.axMachineTimeoutChuckOpen[uiMachine];
	astMachineFaultRequest[uiMachine].xTimeoutChuckClose := GVL_HMI.axMachineTimeoutChuckClose[uiMachine];
	astMachineFaultRequest[uiMachine].xTimeoutCycleStart := GVL_HMI.axMachineTimeoutCycleStart[uiMachine];

	astAxisFaultRequest[uiMachine].xEnabled := GVL_CELL_SETTINGS.xErrorSimulationEnabled;
	astAxisFaultRequest[uiMachine].xJogConflict := GVL_HMI.axSimAxisJogConflict[uiMachine];
END_FOR;

stAxisGroupFaultRequest.xEnabled := GVL_CELL_SETTINGS.xErrorSimulationEnabled;
stAxisGroupFaultRequest.xExecute := GVL_HMI.xSimAxisGroupError;

stRobotFaultRequest.xEnabled := GVL_CELL_SETTINGS.xErrorSimulationEnabled;
stRobotFaultRequest.xWrongAction := GVL_HMI.xSimRobotWrongAction;
stRobotFaultRequest.stGripper.xEnabled := GVL_CELL_SETTINGS.xErrorSimulationEnabled;
stRobotFaultRequest.stGripper.xGripper1Fault := GVL_HMI.xSimGripper1Fault;
stRobotFaultRequest.stGripper.xGripper2Fault := GVL_HMI.xSimGripper2Fault;
stRobotFaultRequest.stGripper.xRotationFault := GVL_HMI.xSimGripperRotationFault;
stRobotFaultRequest.stGripper.xGlobalFault := GVL_HMI.xSimGripperGlobalFault;

stRobotFaultRequest.stPoint.xEnabled := GVL_CELL_SETTINGS.xErrorSimulationEnabled;
stRobotFaultRequest.stPoint.xXOutOfLimit := GVL_HMI.xSimPointXOutOfLimit;
stRobotFaultRequest.stPoint.xYOutOfLimit := GVL_HMI.xSimPointYOutOfLimit;
stRobotFaultRequest.stPoint.xZOutOfLimit := GVL_HMI.xSimPointZOutOfLimit;
stRobotFaultRequest.stPoint.xInvalidVelocity := GVL_HMI.xSimPointInvalidVelocity;

IF NOT GVL_CELL_SETTINGS.xErrorSimulationEnabled THEN
	adwTestMagazineFaultMask[1] := DWORD#0;
	adwTestMagazineFaultMask[2] := DWORD#0;
END_IF;
astMagazineFaultRequest[1].xEnabled := GVL_CELL_SETTINGS.xErrorSimulationEnabled;
astMagazineFaultRequest[1].xWrongOperation := GVL_HMI.xSimMagazineWrongOperation
	OR ((adwTestMagazineFaultMask[1] AND DWORD#16#0000_0001) <> DWORD#0);
astMagazineFaultRequest[1].xNoBlank := GVL_HMI.xSimMagazineNoBlank
	OR ((adwTestMagazineFaultMask[1] AND DWORD#16#0000_0002) <> DWORD#0);
astMagazineFaultRequest[1].xNoFreeSlot := GVL_HMI.xSimMagazineNoFreeSlot
	OR ((adwTestMagazineFaultMask[1] AND DWORD#16#0000_0004) <> DWORD#0);
astMagazineFaultRequest[1].xInvalidSlot := GVL_HMI.xSimMagazineInvalidSlot
	OR ((adwTestMagazineFaultMask[1] AND DWORD#16#0000_0008) <> DWORD#0);
astMagazineFaultRequest[1].xSlotContent := GVL_HMI.xSimMagazineSlotContent
	OR ((adwTestMagazineFaultMask[1] AND DWORD#16#0000_0010) <> DWORD#0);
astMagazineFaultRequest[1].xGeometry := GVL_HMI.xSimMagazineGeometry
	OR ((adwTestMagazineFaultMask[1] AND DWORD#16#0000_0020) <> DWORD#0);
astMagazineFaultRequest[2].xEnabled := GVL_CELL_SETTINGS.xErrorSimulationEnabled
	AND (adwTestMagazineFaultMask[2] <> DWORD#0);
astMagazineFaultRequest[2].xWrongOperation :=
	(adwTestMagazineFaultMask[2] AND DWORD#16#0000_0001) <> DWORD#0;
astMagazineFaultRequest[2].xNoBlank :=
	(adwTestMagazineFaultMask[2] AND DWORD#16#0000_0002) <> DWORD#0;
astMagazineFaultRequest[2].xNoFreeSlot :=
	(adwTestMagazineFaultMask[2] AND DWORD#16#0000_0004) <> DWORD#0;
astMagazineFaultRequest[2].xInvalidSlot :=
	(adwTestMagazineFaultMask[2] AND DWORD#16#0000_0008) <> DWORD#0;
astMagazineFaultRequest[2].xSlotContent :=
	(adwTestMagazineFaultMask[2] AND DWORD#16#0000_0010) <> DWORD#0;
astMagazineFaultRequest[2].xGeometry :=
	(adwTestMagazineFaultMask[2] AND DWORD#16#0000_0020) <> DWORD#0;

stCellFaultRequest.xEnabled := GVL_CELL_SETTINGS.xErrorSimulationEnabled;
stCellFaultRequest.xBothGrippers := GVL_HMI.xSimCellBothGrippers;

stSafetyFaultRequest.xEnabled := GVL_CELL_SETTINGS.xErrorSimulationEnabled;
FOR uiMachine := UINT#1 TO UINT#4 DO
	stSafetyFaultRequest.axEmergencyStopStation[uiMachine] :=
		GVL_HMI.axSimSafetyEmergencyStopStation[uiMachine];
	stSafetyFaultRequest.axDoorUnlocked[uiMachine] :=
		GVL_HMI.axSimSafetyDoorUnlocked[uiMachine];
END_FOR;
FOR uiMachine := UINT#1 TO UINT#2 DO
	stSafetyFaultRequest.axEmergencyStopCabinet[uiMachine] :=
		GVL_HMI.axSimSafetyEmergencyStopCabinet[uiMachine];
END_FOR;
stSafetyFaultRequest.xEmergencyStopMpg := GVL_HMI.xSimSafetyEmergencyStopMpg;
stSafetyFaultRequest.xPhaseRelayFault := GVL_HMI.xSimSafetyPhaseRelayFault;
stSafetyFaultRequest.xPressureRelayFault := GVL_HMI.xSimSafetyPressureRelayFault;
stSafetyFaultRequest.xSafetyRelayFault := GVL_HMI.xSimSafetyRelayFault;

(* ---- PLC_PRG.RunAlarms.st ---- *)
METHOD PRIVATE RunAlarms

// --- BEGIN IMPLEMENTATION ---

// Единая кнопка подсвечивается только тогда, когда существует хотя бы одна авария
// и каждый активный владелец общей команды готов принять тот же импульс сброса.
// Диагностические защёлки симуляторов станков сюда не входят: они обслуживаются
// отдельной командой «Сброс симулятора» на экране инъекций.
xAlarmResetRequired := GVL_CELL_MANAGER.Status.xError
	OR (CELL_SAFETY.Error.dwAlarmActive <> DWORD#0)
	OR GVL_ROBOT.Status.xError
	OR GVL_MACHINE.Status[1].xError
	OR GVL_MACHINE.Status[2].xError
	OR GVL_MACHINE.Status[3].xError
	OR GVL_MAGAZINE.astStatus[1].xError
	OR GVL_MAGAZINE.astStatus[2].xError
	OR (NOT GVL_HMI.xModbusMode AND GVL_AXIS.arrAxis[1].Status.xError)
	OR (NOT GVL_HMI.xModbusMode AND GVL_AXIS.arrAxis[2].Status.xError)
	OR (NOT GVL_HMI.xModbusMode AND GVL_AXIS.arrAxis[3].Status.xError)
	OR (NOT GVL_HMI.xModbusMode AND GVL_AXIS_GROUP.AxisGroup.Status.xLocalError)
	OR (NOT GVL_HMI.xModbusMode AND GVL_AXIS_GROUP.AxisGroup.Status.xLogicalError)
	OR (NOT GVL_HMI.xModbusMode AND GVL_AXIS_GROUP.AxisGroup.Status.xGroupError)
	OR (NOT GVL_HMI.xModbusMode AND (GVL_MOTION_MANAGER.stMotionManager.Error.dwAlarmActive <> DWORD#0))
	OR (NOT GVL_HMI.xModbusMode AND (GVL_POINT_MANAGER.PointManager.Error.dwAlarmActive <> DWORD#0))
	OR (NOT GVL_HMI.xModbusMode AND (GVL_ROBOT.GripperError.dwAlarmActive <> DWORD#0));

xAlarmResetAllowed := ((GVL_TWO_PALLET.uiMode = 0) OR ((NOT GVL_TWO_PALLET.astStatus[1].xError OR GVL_TWO_PALLET.astStatus[1].xResetAllowed) AND (NOT GVL_TWO_PALLET.astStatus[2].xError OR GVL_TWO_PALLET.astStatus[2].xResetAllowed))) AND xAlarmResetRequired
	AND (CELL_SAFETY.Error.dwAlarmActive = DWORD#0)
	AND (NOT GVL_CELL_MANAGER.Status.xError OR GVL_CELL_MANAGER.Status.xResetAllowed)
	AND (NOT GVL_ROBOT.Status.xError OR GVL_ROBOT.Status.xResetAllowed)
	AND (NOT GVL_MACHINE.Status[1].xError OR GVL_MACHINE.Status[1].xResetAllowed)
	AND (NOT GVL_MACHINE.Status[2].xError OR GVL_MACHINE.Status[2].xResetAllowed)
	AND (NOT GVL_MACHINE.Status[3].xError OR GVL_MACHINE.Status[3].xResetAllowed)
	AND (NOT GVL_MAGAZINE.astPartStatus[1].xError
		OR (GVL_MAGAZINE.astError[1].dwAlarmActive = DWORD#0)
		OR fbMagazine1.FaultStatus.xResetAllowed)
	AND (NOT GVL_MAGAZINE.astPartStatus[2].xError
		OR (GVL_MAGAZINE.astError[2].dwAlarmActive = DWORD#0)
		OR fbMagazine2.FaultStatus.xResetAllowed)
	AND (GVL_HMI.xModbusMode OR NOT GVL_AXIS.arrAxis[1].Status.xError OR AXIS_X.FaultStatus.xResetAllowed)
	AND (GVL_HMI.xModbusMode OR NOT GVL_AXIS.arrAxis[2].Status.xError OR AXIS_Y.FaultStatus.xResetAllowed)
	AND (GVL_HMI.xModbusMode OR NOT GVL_AXIS.arrAxis[3].Status.xError OR AXIS_Z.FaultStatus.xResetAllowed)
	AND (GVL_HMI.xModbusMode OR NOT (GVL_AXIS_GROUP.AxisGroup.Status.xLocalError
		OR GVL_AXIS_GROUP.AxisGroup.Status.xLogicalError
		OR GVL_AXIS_GROUP.AxisGroup.Status.xGroupError)
		OR GROUP_XYZ.FaultStatus.xResetAllowed)
	AND (GVL_HMI.xModbusMode OR (GVL_MOTION_MANAGER.stMotionManager.Error.dwAlarmActive = DWORD#0)
		OR GVL_ROBOT.Status.xResetAllowed)
	AND (GVL_HMI.xModbusMode OR (GVL_POINT_MANAGER.PointManager.Error.dwAlarmActive = DWORD#0)
		OR (GVL_ROBOT.Status.xResetAllowed AND ROBOT.FaultStatus.stPoint.xResetAllowed))
	AND (GVL_HMI.xModbusMode OR (GVL_ROBOT.GripperError.dwAlarmActive = DWORD#0)
		OR (GVL_ROBOT.Status.xResetAllowed AND ROBOT.FaultStatus.stGripper.xResetAllowed));

// Два владельца предупреждений используют один источник журнала и общий счётчик.
FOR uiTwin := 1 TO 2 DO
	IF GVL_MAGAZINE.astDiag[uiTwin].stWarning.udiSequence <> audiPartWarningSeen[uiTwin] THEN
		audiPartWarningSeen[uiTwin] := GVL_MAGAZINE.astDiag[uiTwin].stWarning.udiSequence;
		astMagazineWarningMerged[uiTwin].uiCode := GVL_MAGAZINE.astDiag[uiTwin].stWarning.uiCode;
		astMagazineWarningMerged[uiTwin].udiSequence := astMagazineWarningMerged[uiTwin].udiSequence + 1;
	END_IF;
	IF GVL_TWO_PALLET.astDiag[uiTwin].stWarning.udiSequence <> audiTwinWarningSeen[uiTwin] THEN
		audiTwinWarningSeen[uiTwin] := GVL_TWO_PALLET.astDiag[uiTwin].stWarning.udiSequence;
		astMagazineWarningMerged[uiTwin].uiCode := GVL_TWO_PALLET.astDiag[uiTwin].stWarning.uiCode;
		astMagazineWarningMerged[uiTwin].udiSequence := astMagazineWarningMerged[uiTwin].udiSequence + 1;
	END_IF;
END_FOR;

// В журнал передаются все активные ошибки и предупреждения каждого функционального блока.
astAlarmSource[1].eSource := E_ALARM_SOURCE.CELL;
astAlarmSource[1].dwAlarmActive := GVL_CELL_MANAGER.Error.dwAlarmActive;
astAlarmSource[1].xRobotStopRequired := FALSE;
astAlarmSource[1].xGlobalError := GVL_CELL_CONTROL.xGlobalError;
astAlarmSource[1].stWarning := GVL_CELL_MANAGER.Diag.stWarning;

astAlarmSource[2].eSource := E_ALARM_SOURCE.ROBOT;
astAlarmSource[2].dwAlarmActive := GVL_ROBOT.Error.dwAlarmActive;
astAlarmSource[2].xRobotStopRequired := FALSE;
astAlarmSource[2].xGlobalError := GVL_CELL_CONTROL.xGlobalError;
astAlarmSource[2].stWarning := GVL_ROBOT.Diag.stWarning;

astAlarmSource[3].eSource := E_ALARM_SOURCE.MACHINE_1;
astAlarmSource[3].dwAlarmActive := GVL_MACHINE.Error[1].dwAlarmActive;
astAlarmSource[3].xRobotStopRequired := GVL_MACHINE.Status[1].xCriticalError;
astAlarmSource[3].xGlobalError := GVL_CELL_CONTROL.xGlobalError;
astAlarmSource[3].stWarning := GVL_MACHINE.Diag[1].stWarning;

astAlarmSource[4].eSource := E_ALARM_SOURCE.MACHINE_2;
astAlarmSource[4].dwAlarmActive := GVL_MACHINE.Error[2].dwAlarmActive;
astAlarmSource[4].xRobotStopRequired := GVL_MACHINE.Status[2].xCriticalError;
astAlarmSource[4].xGlobalError := GVL_CELL_CONTROL.xGlobalError;
astAlarmSource[4].stWarning := GVL_MACHINE.Diag[2].stWarning;

astAlarmSource[5].eSource := E_ALARM_SOURCE.MACHINE_3;
astAlarmSource[5].dwAlarmActive := GVL_MACHINE.Error[3].dwAlarmActive;
astAlarmSource[5].xRobotStopRequired := GVL_MACHINE.Status[3].xCriticalError;
astAlarmSource[5].xGlobalError := GVL_CELL_CONTROL.xGlobalError;
astAlarmSource[5].stWarning := GVL_MACHINE.Diag[3].stWarning;

astAlarmSource[6].eSource := E_ALARM_SOURCE.MAGAZINE_LOGIC_1;
astAlarmSource[6].dwAlarmActive := GVL_MAGAZINE.astError[1].dwAlarmActive;
astAlarmSource[6].xRobotStopRequired := GVL_MAGAZINE.astStatus[1].xRobotStopRequired;
astAlarmSource[6].xGlobalError := GVL_CELL_CONTROL.xGlobalError;
astAlarmSource[6].stWarning := astMagazineWarningMerged[1];

astAlarmSource[7].eSource := E_ALARM_SOURCE.MAGAZINE_LOGIC_2;
astAlarmSource[7].dwAlarmActive := GVL_MAGAZINE.astError[2].dwAlarmActive;
astAlarmSource[7].xRobotStopRequired := GVL_MAGAZINE.astStatus[2].xRobotStopRequired;
astAlarmSource[7].xGlobalError := GVL_CELL_CONTROL.xGlobalError;
astAlarmSource[7].stWarning := astMagazineWarningMerged[2];

// Числовые коды 7 и 8 зарезервированы, чтобы старые записи SQLite не начали
// отображаться как аварии осей X/Y после удаления приводов магазинов.
astAlarmSource[8].eSource := E_ALARM_SOURCE.RESERVED_LEGACY_MAGAZINE_AXIS_1;
astAlarmSource[8].dwAlarmActive := DWORD#0;
astAlarmSource[8].xRobotStopRequired := FALSE;
astAlarmSource[8].xGlobalError := GVL_CELL_CONTROL.xGlobalError;
astAlarmSource[8].stWarning.uiCode := UINT#0;
astAlarmSource[8].stWarning.udiSequence := UDINT#0;

astAlarmSource[9].eSource := E_ALARM_SOURCE.RESERVED_LEGACY_MAGAZINE_AXIS_2;
astAlarmSource[9].dwAlarmActive := DWORD#0;
astAlarmSource[9].xRobotStopRequired := FALSE;
astAlarmSource[9].xGlobalError := GVL_CELL_CONTROL.xGlobalError;
astAlarmSource[9].stWarning.uiCode := UINT#0;
astAlarmSource[9].stWarning.udiSequence := UDINT#0;

astAlarmSource[10].eSource := E_ALARM_SOURCE.AXIS_X;
IF GVL_HMI.xModbusMode THEN astAlarmSource[10].dwAlarmActive := DWORD#0;
ELSE astAlarmSource[10].dwAlarmActive := GVL_AXIS.arrAxis[1].Error.dwAlarmActive; END_IF;
astAlarmSource[10].xRobotStopRequired := FALSE;
astAlarmSource[10].xGlobalError := GVL_CELL_CONTROL.xGlobalError;
astAlarmSource[10].stWarning := GVL_AXIS.arrAxis[1].Diag.stWarning;

astAlarmSource[11].eSource := E_ALARM_SOURCE.AXIS_Y;
IF GVL_HMI.xModbusMode THEN astAlarmSource[11].dwAlarmActive := DWORD#0;
ELSE astAlarmSource[11].dwAlarmActive := GVL_AXIS.arrAxis[2].Error.dwAlarmActive; END_IF;
astAlarmSource[11].xRobotStopRequired := FALSE;
astAlarmSource[11].xGlobalError := GVL_CELL_CONTROL.xGlobalError;
astAlarmSource[11].stWarning := GVL_AXIS.arrAxis[2].Diag.stWarning;

astAlarmSource[12].eSource := E_ALARM_SOURCE.AXIS_Z;
IF GVL_HMI.xModbusMode THEN astAlarmSource[12].dwAlarmActive := DWORD#0;
ELSE astAlarmSource[12].dwAlarmActive := GVL_AXIS.arrAxis[3].Error.dwAlarmActive; END_IF;
astAlarmSource[12].xRobotStopRequired := FALSE;
astAlarmSource[12].xGlobalError := GVL_CELL_CONTROL.xGlobalError;
astAlarmSource[12].stWarning := GVL_AXIS.arrAxis[3].Diag.stWarning;

astAlarmSource[13].eSource := E_ALARM_SOURCE.AXIS_GROUP;
IF GVL_HMI.xModbusMode THEN astAlarmSource[13].dwAlarmActive := DWORD#0;
ELSE astAlarmSource[13].dwAlarmActive := GVL_AXIS_GROUP.AxisGroup.Error.dwAlarmActive; END_IF;
astAlarmSource[13].xRobotStopRequired := FALSE;
astAlarmSource[13].xGlobalError := GVL_CELL_CONTROL.xGlobalError;
astAlarmSource[13].stWarning := GVL_AXIS_GROUP.AxisGroup.Diag.stWarning;

astAlarmSource[14].eSource := E_ALARM_SOURCE.MOTION_MANAGER;
IF GVL_HMI.xModbusMode THEN astAlarmSource[14].dwAlarmActive := DWORD#0;
ELSE astAlarmSource[14].dwAlarmActive := GVL_MOTION_MANAGER.stMotionManager.Error.dwAlarmActive; END_IF;
astAlarmSource[14].xRobotStopRequired := FALSE;
astAlarmSource[14].xGlobalError := GVL_CELL_CONTROL.xGlobalError;
astAlarmSource[14].stWarning := GVL_MOTION_MANAGER.stMotionManager.Diag.stWarning;

astAlarmSource[15].eSource := E_ALARM_SOURCE.POINT_MANAGER;
IF GVL_HMI.xModbusMode THEN astAlarmSource[15].dwAlarmActive := DWORD#0;
ELSE astAlarmSource[15].dwAlarmActive := GVL_POINT_MANAGER.PointManager.Error.dwAlarmActive; END_IF;
astAlarmSource[15].xRobotStopRequired := FALSE;
astAlarmSource[15].xGlobalError := GVL_CELL_CONTROL.xGlobalError;
astAlarmSource[15].stWarning := GVL_POINT_MANAGER.PointManager.Diag.stWarning;

astAlarmSource[16].eSource := E_ALARM_SOURCE.GRIPPER;
IF GVL_HMI.xModbusMode THEN astAlarmSource[16].dwAlarmActive := DWORD#0;
ELSE astAlarmSource[16].dwAlarmActive := GVL_ROBOT.GripperError.dwAlarmActive; END_IF;
astAlarmSource[16].xRobotStopRequired := FALSE;
astAlarmSource[16].xGlobalError := GVL_CELL_CONTROL.xGlobalError;
astAlarmSource[16].stWarning := GVL_ROBOT.GripperDiag.stWarning;

astAlarmSource[17].eSource := E_ALARM_SOURCE.CELL_SAFETY;
astAlarmSource[17].dwAlarmActive := CELL_SAFETY.Error.dwAlarmActive;
astAlarmSource[17].xRobotStopRequired := TRUE;
astAlarmSource[17].xGlobalError := CELL_SAFETY.Status.xGlobalError;
astAlarmSource[17].stWarning := CELL_SAFETY.Diag.stWarning;

ALARM_MANAGER(
	xResetWarnings := GVL_ALARM.Command.xResetWarnings,
	Sources := astAlarmSource,
	Status => GVL_ALARM.Status,
	Events => GVL_ALARM.Events
);

(* ---- PLC_PRG.RunCellControl.st ---- *)
METHOD PRIVATE RunCellControl

// --- BEGIN IMPLEMENTATION ---

uiMagazine := GVL_CELL_MANAGER.Status.uiActiveMagazine;
IF (uiMagazine < UINT#1) OR (uiMagazine > UINT#2) THEN
	uiMagazine := UINT#1;
END_IF;

TYPE_CONFIG(
	xTestInitialize := xTestInitializePulse,
	stTestScenario := GVL_HMI.stTestScenario,
	Command := GVL_HMI.stMultiType.Command,
	xCellRunning := GVL_CELL_MANAGER.Status.xRunning,
	xMotionBusy := xMotionBusy,
	stRobotStatus := GVL_ROBOT.Status,
	astMagazineStatus := GVL_MAGAZINE.astStatus,
	astMachineStatus := GVL_MACHINE.Status,
	uiRows := GVL_CELL_SETTINGS.MagazineRows,
	uiColumns := GVL_CELL_SETTINGS.MagazineColumns,
	Config => GVL_MULTI_TYPE.Config,
	Status => GVL_MULTI_TYPE.ConfigStatus
);

CELL_MANAGER(
	xStart := GVL_CELL_CONTROL.xStart,
	xStop := GVL_CELL_CONTROL.xStop,
	xTestAbort := xTestAbortActive,
	xResetRequest := GVL_HMI.xCellReset,
	xReset := GVL_CELL_CONTROL.xReset,
	xOperatorChoice := GVL_HMI.xCellOperatorChoice,
	xOperatorCancel := GVL_HMI.xCellOperatorCancel,
	uiOperatorChoice := GVL_HMI.uiCellOperatorChoice,
	xManual := GVL_CELL_CONTROL.xManual,
	uiModeRejectReason := uiCellModeRejectReason,
	xSettingsRejected := xCellSettingRejected,
	xGlobalError := GVL_CELL_CONTROL.xGlobalError,
	xSafetyReady := CELL_SAFETY.Status.xReady,
	xDrivesReady := xDrivesReady,
	xMotionBusy := xMotionBusy,
	xRobotInterfaceReady := xRobotInterfaceReady,
	lrRobotActualX := lrRobotActualX,
	lrRobotActualY := lrRobotActualY,
	lrRobotActualZ := lrRobotActualZ,
	stSafetyHomePoint := GVL_POINT.Points[E_POINT_NAME.HOME_SAFETY],
	lrSafetyHomeToleranceX := GVL_CELL_SETTINGS.lrSafetyHomeToleranceX,
	lrSafetyHomeToleranceY := GVL_CELL_SETTINGS.lrSafetyHomeToleranceY,
	lrSafetyHomeToleranceZ := GVL_CELL_SETTINGS.lrSafetyHomeToleranceZ,
	lrStoppedPoseTolerance := GVL_CELL_SETTINGS.lrStoppedPoseTolerance,
	Config := GVL_MULTI_TYPE.Config,
	xConfigurationValid := GVL_MULTI_TYPE.ConfigStatus.xConfigurationValid,
	xPointsConfigured := xPointTableReady,
	stRobotStatus := GVL_ROBOT.Status,
	astMagazineStatus := GVL_MAGAZINE.astStatus,
	astMachineStatus := GVL_MACHINE.Status,
	astMachineDiag := GVL_MACHINE.Diag,
	FaultRequest := stCellFaultRequest,
	Command => GVL_CELL_MANAGER.Command,
	Status => GVL_CELL_MANAGER.Status,
	Diag => GVL_CELL_MANAGER.Diag,
	Error => GVL_CELL_MANAGER.Error,
	CycleStatus => GVL_MULTI_TYPE.CycleStatus
);

IF GVL_MULTI_TYPE.ConfigStatus.stWarning.udiSequence
<> udiLastTypeConfigWarningSequence THEN
	GVL_CELL_MANAGER.Diag.stWarning := GVL_MULTI_TYPE.ConfigStatus.stWarning;
	udiLastTypeConfigWarningSequence := GVL_MULTI_TYPE.ConfigStatus.stWarning.udiSequence;
END_IF;

// Сначала снимаем команды обоих владельцев, затем маршрутизируем единственную
// команду менеджера выбранному магазину.
FOR uiMagazine := UINT#1 TO UINT#2 DO
	GVL_MAGAZINE.astAutoCommand[uiMagazine].xEnable := FALSE;
	GVL_MAGAZINE.astAutoCommand[uiMagazine].xDisable := GVL_CELL_CONTROL.xDisable;
	GVL_MAGAZINE.astAutoCommand[uiMagazine].xExecute := FALSE;
	GVL_MAGAZINE.astAutoCommand[uiMagazine].xStop := FALSE;
	GVL_MAGAZINE.astAutoCommand[uiMagazine].eOperation := E_MAGAZINE_OPERATION.NONE;
	GVL_MAGAZINE.astAutoCommand[uiMagazine].iTakeSlot := SINT#0;
	GVL_MAGAZINE.astAutoCommand[uiMagazine].iPutSlot := SINT#0;
END_FOR;
IF (GVL_CELL_MANAGER.Status.uiActiveMagazine >= UINT#1)
AND (GVL_CELL_MANAGER.Status.uiActiveMagazine <= UINT#2) THEN
	GVL_MAGAZINE.astAutoCommand[GVL_CELL_MANAGER.Status.uiActiveMagazine] :=
		GVL_CELL_MANAGER.Command.stMagazine;
	GVL_MAGAZINE.astAutoCommand[GVL_CELL_MANAGER.Status.uiActiveMagazine].xEnable := FALSE;
	GVL_MAGAZINE.astAutoCommand[GVL_CELL_MANAGER.Status.uiActiveMagazine].xDisable :=
		GVL_CELL_CONTROL.xDisable;
END_IF;

(* ---- PLC_PRG.RunMachines.st ---- *)
METHOD PRIVATE RunMachines

// --- BEGIN IMPLEMENTATION ---

// Импульсные команды HMI изменяют сохранённое разрешение работы станка.
FOR uiMachine := 1 TO 3 DO
	IF GVL_HMI.axMachineDisable[uiMachine] THEN
		GVL_HMI.axMachineUsed[uiMachine] := FALSE;
	ELSIF GVL_HMI.axMachineEnable[uiMachine] THEN
		GVL_HMI.axMachineUsed[uiMachine] := TRUE;
	END_IF;
END_FOR;

MACHINE_1.stPoints.eAbove := E_POINT_NAME.MACHINE_1_ABOVE;
MACHINE_1.stPoints.eChuck := E_POINT_NAME.MACHINE_1_CHUCK_POSITION;
MACHINE_1.stPoints.eChuckApproach := E_POINT_NAME.MACHINE_1_CHUCK_APROACH;
MACHINE_1.stPoints.eInside := E_POINT_NAME.MACHINE_1_INSIDE;
MACHINE_1.stPoints.eNone := E_POINT_NAME.NONE;

// Виртуальные устройства исполняют команду предыдущего цикла. Затем слой
// инъекции формирует обратную связь, которую увидит технологический автомат.
MACHINE_1_SIM(
	xTestInitialize := xTestInitializePulse,
	uiTestInitialState := GVL_HMI.stTestScenario.auiMachineState[1],
	xSafetyDoorOpen := GVL_CELL_SETTINGS.xErrorSimulationEnabled
		AND GVL_HMI.axMachineSimSafetyDoorOpen[1],
	Command := GVL_MACHINE.Command[1].stIo,
	FaultRequest := astMachineFaultRequest[1],
	xSimulationAccelerationEnable := GVL_CELL_SETTINGS.xSimulationAccelerationActive,
	uiSimulationTimeFactor := GVL_CELL_SETTINGS.uiSimulationTimeFactorApplied,
	tDoorOpenTime := GVL_HMI.tMachineDoorOpenTime,
	tDoorCloseTime := GVL_HMI.tMachineDoorCloseTime,
	tChuckOpenTime := GVL_HMI.tMachineChuckOpenTime,
	tChuckCloseTime := GVL_HMI.tMachineChuckCloseTime,
	tCycleTime := GVL_HMI.tMachineCycleTime[1]
);
MACHINE_2_SIM(
	xTestInitialize := xTestInitializePulse,
	uiTestInitialState := GVL_HMI.stTestScenario.auiMachineState[2],
	xSafetyDoorOpen := GVL_CELL_SETTINGS.xErrorSimulationEnabled
		AND GVL_HMI.axMachineSimSafetyDoorOpen[2],
	Command := GVL_MACHINE.Command[2].stIo,
	FaultRequest := astMachineFaultRequest[2],
	xSimulationAccelerationEnable := GVL_CELL_SETTINGS.xSimulationAccelerationActive,
	uiSimulationTimeFactor := GVL_CELL_SETTINGS.uiSimulationTimeFactorApplied,
	tDoorOpenTime := GVL_HMI.tMachineDoorOpenTime,
	tDoorCloseTime := GVL_HMI.tMachineDoorCloseTime,
	tChuckOpenTime := GVL_HMI.tMachineChuckOpenTime,
	tChuckCloseTime := GVL_HMI.tMachineChuckCloseTime,
	tCycleTime := GVL_HMI.tMachineCycleTime[2]
);
MACHINE_3_SIM(
	xTestInitialize := xTestInitializePulse,
	uiTestInitialState := GVL_HMI.stTestScenario.auiMachineState[3],
	xSafetyDoorOpen := GVL_CELL_SETTINGS.xErrorSimulationEnabled
		AND GVL_HMI.axMachineSimSafetyDoorOpen[3],
	Command := GVL_MACHINE.Command[3].stIo,
	FaultRequest := astMachineFaultRequest[3],
	xSimulationAccelerationEnable := GVL_CELL_SETTINGS.xSimulationAccelerationActive,
	uiSimulationTimeFactor := GVL_CELL_SETTINGS.uiSimulationTimeFactorApplied,
	tDoorOpenTime := GVL_HMI.tMachineDoorOpenTime,
	tDoorCloseTime := GVL_HMI.tMachineDoorCloseTime,
	tChuckOpenTime := GVL_HMI.tMachineChuckOpenTime,
	tChuckCloseTime := GVL_HMI.tMachineChuckCloseTime,
	tCycleTime := GVL_HMI.tMachineCycleTime[3]
);

MACHINE_1_FAULT(
	Request := astMachineFaultRequest[1],
	MachineStatusRaw := MACHINE_1_SIM.Status,
	RobotStatusRaw := GVL_ROBOT.Status,
	NominalTimeouts := GVL_CELL_SETTINGS.stMachineTimeouts
);
MACHINE_2_FAULT(
	Request := astMachineFaultRequest[2],
	MachineStatusRaw := MACHINE_2_SIM.Status,
	RobotStatusRaw := GVL_ROBOT.Status,
	NominalTimeouts := GVL_CELL_SETTINGS.stMachineTimeouts
);
MACHINE_3_FAULT(
	Request := astMachineFaultRequest[3],
	MachineStatusRaw := MACHINE_3_SIM.Status,
	RobotStatusRaw := GVL_ROBOT.Status,
	NominalTimeouts := GVL_CELL_SETTINGS.stMachineTimeouts
);

MACHINE_1(
	xTestInitialize := xTestInitializePulse,
	uiTestInitialState := GVL_HMI.stTestScenario.auiMachineState[1],
	uiTestProductType := GVL_HMI.stTestScenario.auiMachineType[1],
	xExecute := GVL_CELL_MANAGER.Command.axMachineExecute[1],
	xReset := GVL_HMI.axMachineReset[1],
	xResetGlobal := GVL_CELL_CONTROL.xReset,
	xGlobalError := GVL_CELL_CONTROL.xGlobalError,
	xManualMode := GVL_CELL_CONTROL.xManual,
	xAutomaticUseEnabled := GVL_HMI.axMachineUsed[1],
	xHmiOpenSafetyDoor := GVL_HMI.axMachineManualSafetyDoorOpen[1],
	xHmiCloseSafetyDoor := GVL_HMI.axMachineManualSafetyDoorClose[1],
	xHmiOpenHatch := GVL_HMI.axMachineManualHatchOpen[1],
	xHmiCloseHatch := GVL_HMI.axMachineManualHatchClose[1],
	xHmiOpenChuck := GVL_HMI.axMachineManualChuckOpen[1],
	xHmiCloseChuck := GVL_HMI.axMachineManualChuckClose[1],
	xHmiEnable := GVL_HMI.axMachineEnable[1] AND GVL_HMI.axMachineUsed[1],
	xHmiDisable := GVL_HMI.axMachineDisable[1],
	xHmiSetBlank := GVL_HMI.axMachineSetBlank[1],
	xHmiSetDetail := GVL_HMI.axMachineSetDetail[1],
	xHmiAcceptDoor := GVL_HMI.axMachineAcceptDoor[1],
	xHmiRejectDoor := GVL_HMI.axMachineRejectDoor[1],
	xHmiAcceptRunCNC := GVL_HMI.axMachineAcceptRun[1],
	xHmiRejectRunCNC := GVL_HMI.axMachineRejectRun[1],
	xUseHmiCycleTime := GVL_HMI.xUseHmiCycleTime[1],
	tHmiCycleTime := GVL_HMI.tMachineCycleTime[1],
	stTimeouts := MACHINE_1_FAULT.Timeouts,
	stChangeRecipe := GVL_CELL_SETTINGS.CHANGE_MACHINE,
	stLoadRecipe := GVL_CELL_SETTINGS.LOAD_MACHINE,
	stUnloadRecipe := GVL_CELL_SETTINGS.UNLOAD_MACHINE,
	stMachineStatus := MACHINE_1_FAULT.MachineStatus,
	stRobotStatus := MACHINE_1_FAULT.RobotStatus,
	eRobotTargetPoint := GVL_ROBOT.Diag.eActivePoint,
	xRobotMotionBusy := xMotionBusy,
	Command => GVL_MACHINE.Command[1],
	Status => GVL_MACHINE.Status[1],
	Diag => GVL_MACHINE.Diag[1],
	Error => GVL_MACHINE.Error[1]
);

MACHINE_2.stPoints.eAbove := E_POINT_NAME.MACHINE_2_ABOVE;
MACHINE_2.stPoints.eChuck := E_POINT_NAME.MACHINE_2_CHUCK_POSITION;
MACHINE_2.stPoints.eChuckApproach := E_POINT_NAME.MACHINE_2_CHUCK_APROACH;
MACHINE_2.stPoints.eInside := E_POINT_NAME.MACHINE_2_INSIDE;
MACHINE_2.stPoints.eNone := E_POINT_NAME.NONE;

MACHINE_2(
	xTestInitialize := xTestInitializePulse,
	uiTestInitialState := GVL_HMI.stTestScenario.auiMachineState[2],
	uiTestProductType := GVL_HMI.stTestScenario.auiMachineType[2],
	xExecute := GVL_CELL_MANAGER.Command.axMachineExecute[2],
	xReset := GVL_HMI.axMachineReset[2],
	xResetGlobal := GVL_CELL_CONTROL.xReset,
	xGlobalError := GVL_CELL_CONTROL.xGlobalError,
	xManualMode := GVL_CELL_CONTROL.xManual,
	xAutomaticUseEnabled := GVL_HMI.axMachineUsed[2],
	xHmiOpenSafetyDoor := GVL_HMI.axMachineManualSafetyDoorOpen[2],
	xHmiCloseSafetyDoor := GVL_HMI.axMachineManualSafetyDoorClose[2],
	xHmiOpenHatch := GVL_HMI.axMachineManualHatchOpen[2],
	xHmiCloseHatch := GVL_HMI.axMachineManualHatchClose[2],
	xHmiOpenChuck := GVL_HMI.axMachineManualChuckOpen[2],
	xHmiCloseChuck := GVL_HMI.axMachineManualChuckClose[2],
	xHmiEnable := GVL_HMI.axMachineEnable[2] AND GVL_HMI.axMachineUsed[2],
	xHmiDisable := GVL_HMI.axMachineDisable[2],
	xHmiSetBlank := GVL_HMI.axMachineSetBlank[2],
	xHmiSetDetail := GVL_HMI.axMachineSetDetail[2],
	xHmiAcceptDoor := GVL_HMI.axMachineAcceptDoor[2],
	xHmiRejectDoor := GVL_HMI.axMachineRejectDoor[2],
	xHmiAcceptRunCNC := GVL_HMI.axMachineAcceptRun[2],
	xHmiRejectRunCNC := GVL_HMI.axMachineRejectRun[2],
	xUseHmiCycleTime := GVL_HMI.xUseHmiCycleTime[2],
	tHmiCycleTime := GVL_HMI.tMachineCycleTime[2],
	stTimeouts := MACHINE_2_FAULT.Timeouts,
	stChangeRecipe := GVL_CELL_SETTINGS.CHANGE_MACHINE,
	stLoadRecipe := GVL_CELL_SETTINGS.LOAD_MACHINE,
	stUnloadRecipe := GVL_CELL_SETTINGS.UNLOAD_MACHINE,
	stMachineStatus := MACHINE_2_FAULT.MachineStatus,
	stRobotStatus := MACHINE_2_FAULT.RobotStatus,
	eRobotTargetPoint := GVL_ROBOT.Diag.eActivePoint,
	xRobotMotionBusy := xMotionBusy,
	Command => GVL_MACHINE.Command[2],
	Status => GVL_MACHINE.Status[2],
	Diag => GVL_MACHINE.Diag[2],
	Error => GVL_MACHINE.Error[2]
);

MACHINE_3.stPoints.eAbove := E_POINT_NAME.MACHINE_3_ABOVE;
MACHINE_3.stPoints.eChuck := E_POINT_NAME.MACHINE_3_CHUCK_POSITION;
MACHINE_3.stPoints.eChuckApproach := E_POINT_NAME.MACHINE_3_CHUCK_APROACH;
MACHINE_3.stPoints.eInside := E_POINT_NAME.MACHINE_3_INSIDE;
MACHINE_3.stPoints.eNone := E_POINT_NAME.NONE;

MACHINE_3(
	xTestInitialize := xTestInitializePulse,
	uiTestInitialState := GVL_HMI.stTestScenario.auiMachineState[3],
	uiTestProductType := GVL_HMI.stTestScenario.auiMachineType[3],
	xExecute := GVL_CELL_MANAGER.Command.axMachineExecute[3],
	xReset := GVL_HMI.axMachineReset[3],
	xResetGlobal := GVL_CELL_CONTROL.xReset,
	xGlobalError := GVL_CELL_CONTROL.xGlobalError,
	xManualMode := GVL_CELL_CONTROL.xManual,
	xAutomaticUseEnabled := GVL_HMI.axMachineUsed[3],
	xHmiOpenSafetyDoor := GVL_HMI.axMachineManualSafetyDoorOpen[3],
	xHmiCloseSafetyDoor := GVL_HMI.axMachineManualSafetyDoorClose[3],
	xHmiOpenHatch := GVL_HMI.axMachineManualHatchOpen[3],
	xHmiCloseHatch := GVL_HMI.axMachineManualHatchClose[3],
	xHmiOpenChuck := GVL_HMI.axMachineManualChuckOpen[3],
	xHmiCloseChuck := GVL_HMI.axMachineManualChuckClose[3],
	xHmiEnable := GVL_HMI.axMachineEnable[3] AND GVL_HMI.axMachineUsed[3],
	xHmiDisable := GVL_HMI.axMachineDisable[3],
	xHmiSetBlank := GVL_HMI.axMachineSetBlank[3],
	xHmiSetDetail := GVL_HMI.axMachineSetDetail[3],
	xHmiAcceptDoor := GVL_HMI.axMachineAcceptDoor[3],
	xHmiRejectDoor := GVL_HMI.axMachineRejectDoor[3],
	xHmiAcceptRunCNC := GVL_HMI.axMachineAcceptRun[3],
	xHmiRejectRunCNC := GVL_HMI.axMachineRejectRun[3],
	xUseHmiCycleTime := GVL_HMI.xUseHmiCycleTime[3],
	tHmiCycleTime := GVL_HMI.tMachineCycleTime[3],
	stTimeouts := MACHINE_3_FAULT.Timeouts,
	stChangeRecipe := GVL_CELL_SETTINGS.CHANGE_MACHINE,
	stLoadRecipe := GVL_CELL_SETTINGS.LOAD_MACHINE,
	stUnloadRecipe := GVL_CELL_SETTINGS.UNLOAD_MACHINE,
	stMachineStatus := MACHINE_3_FAULT.MachineStatus,
	stRobotStatus := MACHINE_3_FAULT.RobotStatus,
	eRobotTargetPoint := GVL_ROBOT.Diag.eActivePoint,
	xRobotMotionBusy := xMotionBusy,
	Command => GVL_MACHINE.Command[3],
	Status => GVL_MACHINE.Status[3],
	Diag => GVL_MACHINE.Diag[3],
	Error => GVL_MACHINE.Error[3]
);

// Публичный IO-снимок совпадает с обратной связью, которую анализирует FB_MACHINE.
GVL_MACHINE.Status[1].stIo := MACHINE_1_FAULT.MachineStatus;
GVL_MACHINE.Status[2].stIo := MACHINE_2_FAULT.MachineStatus;
GVL_MACHINE.Status[3].stIo := MACHINE_3_FAULT.MachineStatus;

(* ---- PLC_PRG.RunMagazine.st ---- *)
METHOD PRIVATE RunMagazine

// --- BEGIN IMPLEMENTATION ---

auiMagazineEditSlot[1] := GVL_HMI.astMagazineCommand[1].uiEditSlot;
IF auiMagazineEditSlot[1] = UINT#0 THEN
	auiMagazineEditSlot[1] := GVL_HMI.uiMagazineEditSlot;
END_IF;
auiMagazineEditSlot[2] := GVL_HMI.astMagazineCommand[2].uiEditSlot;

fbMagazine1(
	uiMagazineId := UINT#1,
	xMechanismReady := (GVL_TWO_PALLET.uiMode = 0) OR GVL_TWO_PALLET.astStatus[1].xReady,
	xTestInitialize := xTestInitializePulse OR xTestAbortActive,
	xTestEnabled := GVL_HMI.stTestScenario.axMagazineEnabled[1],
	stRobotStatus := GVL_ROBOT.Status,
	astMachineStatus := GVL_MACHINE.Status,
	auiMachineType := GVL_MULTI_TYPE.Config.auiMachineType,
	stMagazineCommand := GVL_MAGAZINE.astAutoCommand[1],
	stHmiCommand := GVL_HMI.stRobotCommand,
	xManual := GVL_CELL_CONTROL.xManual AND NOT GVL_CELL_MANAGER.Status.xRunning,
	xReset := GVL_CELL_CONTROL.xReset OR GVL_HMI.astMagazineCommand[1].xReset OR ((GVL_TWO_PALLET.uiMode = 1) AND (GVL_TWO_PALLET.auiCommand[1] = 16) AND GVL_TWO_PALLET.astStatus[1].xCommandAccepted),
	xGlobalError := GVL_CELL_CONTROL.xGlobalError,
	xHmiEnable := ((GVL_TWO_PALLET.uiMode = 0) AND (GVL_HMI.astMagazineCommand[1].xEnable OR GVL_HMI.xMagazineEnable))
		OR ((GVL_TWO_PALLET.uiMode = 1) AND GVL_TWO_PALLET.astStatus[1].xReady
			AND NOT fbMagazine1.Status.xEnabled AND NOT fbMagazine1.Status.xFinished),
	xHmiDisable := GVL_HMI.astMagazineCommand[1].xDisable OR GVL_HMI.xMagazineDisable OR ((GVL_TWO_PALLET.uiMode = 1) AND (NOT GVL_TWO_PALLET.astStatus[1].xEnabled OR GVL_TWO_PALLET.astStatus[1].xBusy)),
	xHmiFillBlanks := (GVL_TWO_PALLET.uiMode = 0) AND (GVL_HMI.astMagazineCommand[1].xFill OR GVL_HMI.xMagazineFillBlanks),
	xHmiClear := (GVL_TWO_PALLET.uiMode = 0) AND (GVL_HMI.astMagazineCommand[1].xClear OR GVL_HMI.xMagazineClear),
	xHmiCycleSlot := (GVL_TWO_PALLET.uiMode = 0) AND (GVL_HMI.astMagazineCommand[1].xCycleSlot OR GVL_HMI.xMagazineCycleSlot),
	xHmiApplySlot := (GVL_TWO_PALLET.uiMode = 0) AND (GVL_HMI.astMagazineCommand[1].xApplySlot),
	xHmiApplyPitchX := GVL_HMI.astMagazineCommand[1].xApplyPitchX,
	xHmiApplyPitchY := GVL_HMI.astMagazineCommand[1].xApplyPitchY,
	uiHmiEditSlot := auiMagazineEditSlot[1],
	uiHmiEditDetailType := GVL_HMI.astMagazineCommand[1].uiEditDetailType,
	uiHmiEditProductType := GVL_HMI.astMagazineCommand[1].uiEditProductType,
	lrHmiEditPitchX := GVL_HMI.astMagazineCommand[1].lrEditPitchX,
	lrHmiEditPitchY := GVL_HMI.astMagazineCommand[1].lrEditPitchY,
	xRobotOwnsMagazine := (GVL_CELL_MANAGER.Status.uiActiveMagazine = UINT#1)
		AND (GVL_CELL_MANAGER.Status.xRunning OR GVL_ROBOT.Status.xBusy),
	xRobotCanWorkWithMagazine := xRobotInterfaceReady
		AND xPointTableReady
		AND NOT GVL_ROBOT.Status.xError,
	xSharedGeometryEditAllowed := NOT GVL_MAGAZINE.astStatus[1].xEnabled
		AND NOT GVL_MAGAZINE.astStatus[2].xEnabled
		AND NOT GVL_HMI.xMagazineEnable
		AND NOT GVL_HMI.astMagazineCommand[1].xEnable
		AND NOT GVL_HMI.astMagazineCommand[2].xEnable,
	uiRows := GVL_CELL_SETTINGS.MagazineRows,
	uiColumns := GVL_CELL_SETTINGS.MagazineColumns,
	uiTypeCount := GVL_MULTI_TYPE.Config.uiTypeCount,
	auiSlotType := GVL_MULTI_TYPE.Config.auiSlotType,
	FaultRequest := astMagazineFaultRequest[1],
	stInventory := GVL_DETAIL.astMagazine[1],
	lrPitchX := GVL_HMI.MagazinePitchX,
	lrPitchY := GVL_HMI.MagazinePitchY,
	Command => GVL_MAGAZINE.astCommand[1],
	Status => GVL_MAGAZINE.astPartStatus[1],
	Diag => GVL_MAGAZINE.astDiag[1],
	Error => GVL_MAGAZINE.astError[1]
);

fbMagazine2(
	uiMagazineId := UINT#2,
	xMechanismReady := (GVL_TWO_PALLET.uiMode = 0) OR GVL_TWO_PALLET.astStatus[2].xReady,
	xTestInitialize := xTestInitializePulse OR xTestAbortActive,
	xTestEnabled := GVL_HMI.stTestScenario.axMagazineEnabled[2],
	stRobotStatus := GVL_ROBOT.Status,
	astMachineStatus := GVL_MACHINE.Status,
	auiMachineType := GVL_MULTI_TYPE.Config.auiMachineType,
	stMagazineCommand := GVL_MAGAZINE.astAutoCommand[2],
	stHmiCommand := GVL_HMI.stRobotCommand,
	xManual := GVL_CELL_CONTROL.xManual AND NOT GVL_CELL_MANAGER.Status.xRunning,
	xReset := GVL_CELL_CONTROL.xReset OR GVL_HMI.astMagazineCommand[2].xReset OR ((GVL_TWO_PALLET.uiMode = 1) AND (GVL_TWO_PALLET.auiCommand[2] = 16) AND GVL_TWO_PALLET.astStatus[2].xCommandAccepted),
	xGlobalError := GVL_CELL_CONTROL.xGlobalError,
	xHmiEnable := ((GVL_TWO_PALLET.uiMode = 0) AND (GVL_HMI.astMagazineCommand[2].xEnable))
		OR ((GVL_TWO_PALLET.uiMode = 1) AND GVL_TWO_PALLET.astStatus[2].xReady
			AND NOT fbMagazine2.Status.xEnabled AND NOT fbMagazine2.Status.xFinished),
	xHmiDisable := GVL_HMI.astMagazineCommand[2].xDisable OR ((GVL_TWO_PALLET.uiMode = 1) AND (NOT GVL_TWO_PALLET.astStatus[2].xEnabled OR GVL_TWO_PALLET.astStatus[2].xBusy)),
	xHmiFillBlanks := (GVL_TWO_PALLET.uiMode = 0) AND (GVL_HMI.astMagazineCommand[2].xFill),
	xHmiClear := (GVL_TWO_PALLET.uiMode = 0) AND (GVL_HMI.astMagazineCommand[2].xClear),
	xHmiCycleSlot := (GVL_TWO_PALLET.uiMode = 0) AND (GVL_HMI.astMagazineCommand[2].xCycleSlot),
	xHmiApplySlot := (GVL_TWO_PALLET.uiMode = 0) AND (GVL_HMI.astMagazineCommand[2].xApplySlot),
	xHmiApplyPitchX := GVL_HMI.astMagazineCommand[2].xApplyPitchX,
	xHmiApplyPitchY := GVL_HMI.astMagazineCommand[2].xApplyPitchY,
	uiHmiEditSlot := auiMagazineEditSlot[2],
	uiHmiEditDetailType := GVL_HMI.astMagazineCommand[2].uiEditDetailType,
	uiHmiEditProductType := GVL_HMI.astMagazineCommand[2].uiEditProductType,
	lrHmiEditPitchX := GVL_HMI.astMagazineCommand[2].lrEditPitchX,
	lrHmiEditPitchY := GVL_HMI.astMagazineCommand[2].lrEditPitchY,
	xRobotOwnsMagazine := (GVL_CELL_MANAGER.Status.uiActiveMagazine = UINT#2)
		AND (GVL_CELL_MANAGER.Status.xRunning OR GVL_ROBOT.Status.xBusy),
	xRobotCanWorkWithMagazine := xRobotInterfaceReady
		AND xPointTableReady
		AND NOT GVL_ROBOT.Status.xError,
	xSharedGeometryEditAllowed := NOT GVL_MAGAZINE.astStatus[1].xEnabled
		AND NOT GVL_MAGAZINE.astStatus[2].xEnabled
		AND NOT GVL_HMI.xMagazineEnable
		AND NOT GVL_HMI.astMagazineCommand[1].xEnable
		AND NOT GVL_HMI.astMagazineCommand[2].xEnable,
	uiRows := GVL_CELL_SETTINGS.MagazineRows,
	uiColumns := GVL_CELL_SETTINGS.MagazineColumns,
	uiTypeCount := GVL_MULTI_TYPE.Config.uiTypeCount,
	auiSlotType := GVL_MULTI_TYPE.Config.auiSlotType,
	FaultRequest := astMagazineFaultRequest[2],
	stInventory := GVL_DETAIL.astMagazine[2],
	lrPitchX := GVL_HMI.MagazinePitchX,
	lrPitchY := GVL_HMI.MagazinePitchY,
	Command => GVL_MAGAZINE.astCommand[2],
	Status => GVL_MAGAZINE.astPartStatus[2],
	Diag => GVL_MAGAZINE.astDiag[2],
	Error => GVL_MAGAZINE.astError[2]
);

// Сохранить физический инвентарь текущей палеты после подтверждённых действий робота.
FOR uiTwin := 1 TO 2 DO
	GVL_MAGAZINE.astStatus[uiTwin] := GVL_MAGAZINE.astPartStatus[uiTwin];
	IF NOT GVL_TWO_PALLET.astStatus[uiTwin].xError THEN axTwinRobotStopLatched[uiTwin] := FALSE;
	ELSIF GVL_ROBOT.Status.uiMagazineContext = uiTwin THEN axTwinRobotStopLatched[uiTwin] := TRUE; END_IF;
	IF GVL_TWO_PALLET.uiMode = 1 THEN
		uiTwinPallet := GVL_TWO_PALLET.astStatus[uiTwin].uiRobotPallet;
		IF (uiTwinPallet >= UINT#1) AND (uiTwinPallet <= UINT#2) THEN
			GVL_TWO_PALLET.astStore[uiTwin].astPallet[uiTwinPallet] := GVL_DETAIL.astMagazine[uiTwin];
		END_IF;
		GVL_MAGAZINE.astStatus[uiTwin].xReady := GVL_MAGAZINE.astStatus[uiTwin].xReady AND GVL_TWO_PALLET.astStatus[uiTwin].xReady;
		GVL_MAGAZINE.astStatus[uiTwin].xEnableSequenceAllowed := GVL_TWO_PALLET.astStatus[uiTwin].xEnableAllowed;
		GVL_MAGAZINE.astStatus[uiTwin].xEnabled := GVL_TWO_PALLET.astStatus[uiTwin].xEnabled;
		GVL_MAGAZINE.astStatus[uiTwin].xBusy := GVL_MAGAZINE.astPartStatus[uiTwin].xBusy OR GVL_TWO_PALLET.astStatus[uiTwin].xBusy;
		GVL_MAGAZINE.astStatus[uiTwin].xFillAllowed := FALSE;
		GVL_MAGAZINE.astStatus[uiTwin].xClearAllowed := FALSE;
		GVL_MAGAZINE.astStatus[uiTwin].xEditAllowed := FALSE;
		GVL_MAGAZINE.astStatus[uiTwin].xError := GVL_MAGAZINE.astStatus[uiTwin].xError OR GVL_TWO_PALLET.astStatus[uiTwin].xError;
		GVL_MAGAZINE.astError[uiTwin].dwErrorActive := GVL_MAGAZINE.astError[uiTwin].dwErrorActive
			OR GVL_TWO_PALLET.astError[uiTwin].dwErrorActive;
		GVL_MAGAZINE.astError[uiTwin].dwAlarmActive := GVL_MAGAZINE.astError[uiTwin].dwAlarmActive
			OR GVL_TWO_PALLET.astError[uiTwin].dwAlarmActive;
		GVL_MAGAZINE.astStatus[uiTwin].xRobotStopRequired := GVL_MAGAZINE.astStatus[uiTwin].xRobotStopRequired
			OR axTwinRobotStopLatched[uiTwin];
		IF axTwinRobotStopLatched[uiTwin] THEN
			GVL_MAGAZINE.astCommand[uiTwin].xStop := TRUE;
			GVL_MAGAZINE.astCommand[uiTwin].xExecute := FALSE;
		END_IF;
	ELSE
		GVL_TWO_PALLET.astStatic[uiTwin] := GVL_DETAIL.astMagazine[uiTwin];
	END_IF;
END_FOR;

IF GVL_TWO_PALLET.uiMode = 0 THEN
	GVL_TWO_PALLET.lrStaticPitchX := GVL_HMI.MagazinePitchX;
	GVL_TWO_PALLET.lrStaticPitchY := GVL_HMI.MagazinePitchY;
ELSE
	GVL_TWO_PALLET.lrTwinPitchX := GVL_HMI.MagazinePitchX;
	GVL_TWO_PALLET.lrTwinPitchY := GVL_HMI.MagazinePitchY;
END_IF;
